// TIA Portal V17 export
// export: Created 2021-12-03T08:13:05.5673976Z, ExportSetting WithDefaults, DisplayName Totally Integrated Automation Portal, DisplayVersion V17, DisplayName TIA Portal Openness, DisplayVersion V17, DisplayName TIA Portal Version Control Interface, DisplayVersion V17, DisplayName STEP 7 Professional, DisplayVersion V17, DisplayName STEP 7 Safety, DisplayVersion V17, DisplayName WinCC Advanced, DisplayVersion V17
FUNCTION "FC_SpdClclt" : Void   // FC503, FBD
VERSION : 0.1
// stored: AutoNumber false, IsIECCheckEnabled false, UDAEnableTagReadback false
   VAR_TEMP
      "Time" : Real;
   END_VAR
   VAR_TEMP   // added for the SCL form of the ladder/FBD networks
      _w1 : Bool;
   END_VAR
BEGIN

REGION Network 1: Условие для запуска
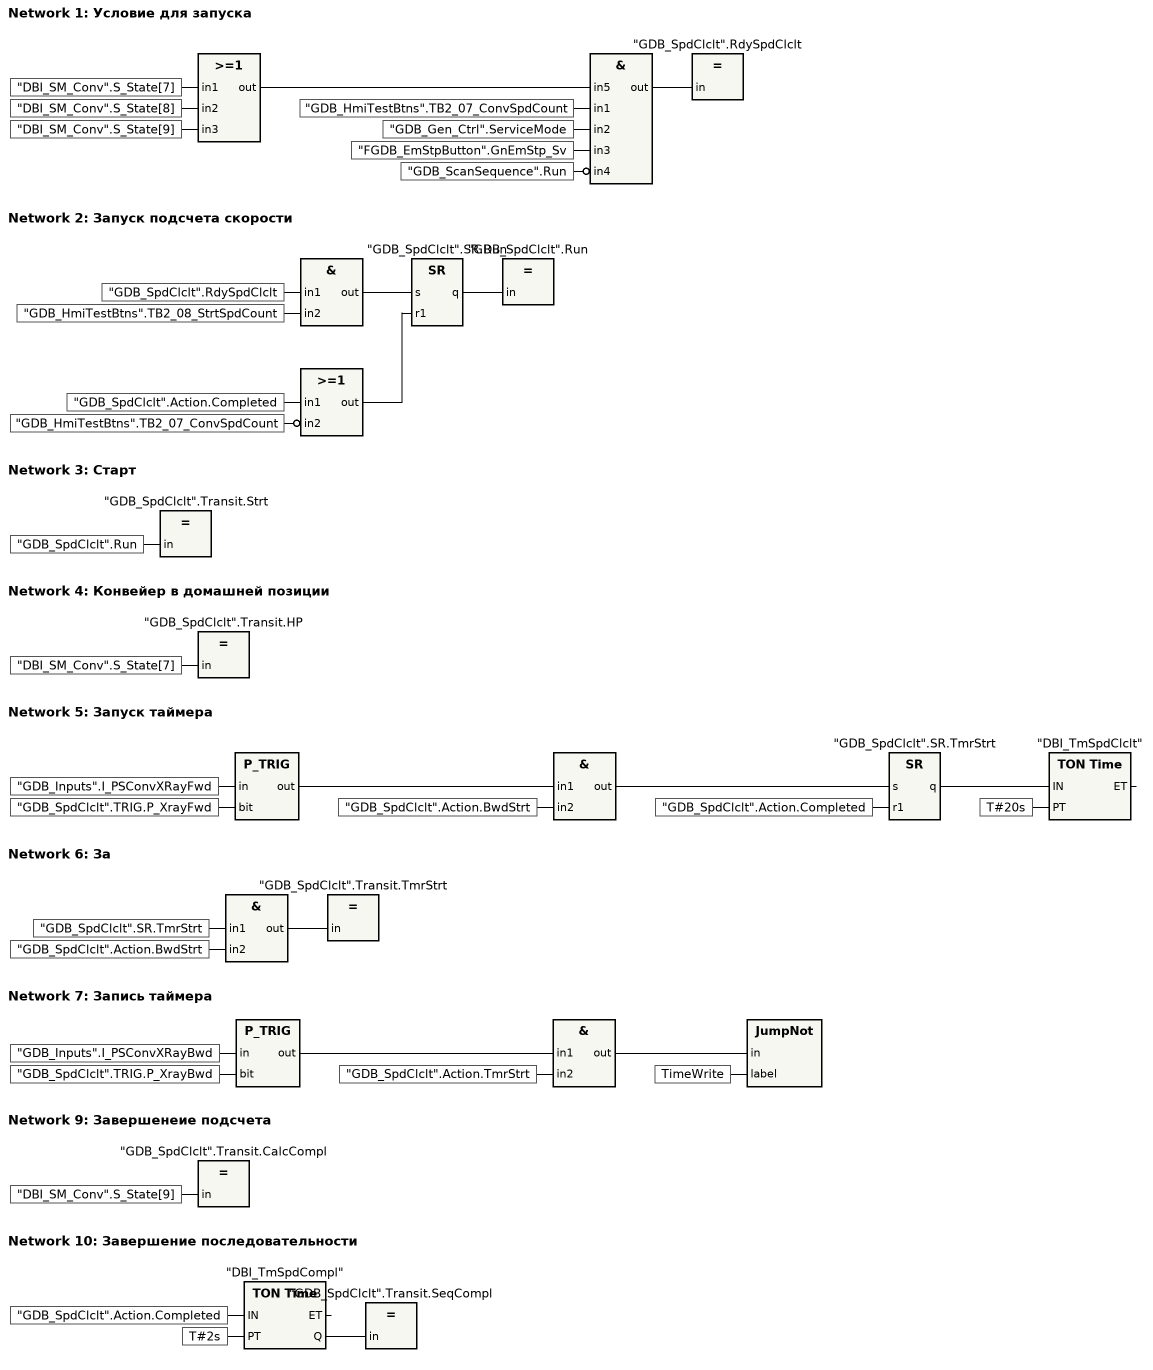
   "GDB_SpdClclt".RdySpdClclt := ("DBI_SM_Conv".S_State[7] OR "DBI_SM_Conv".S_State[8] OR "DBI_SM_Conv".S_State[9]) AND "GDB_HmiTestBtns".TB2_07_ConvSpdCount AND "GDB_Gen_Ctrl".ServiceMode AND "FGDB_EmStpButton".GnEmStp_Sv AND NOT "GDB_ScanSequence".Run;
END_REGION

REGION Network 2: Запуск подсчета скорости
   IF "GDB_SpdClclt".RdySpdClclt AND "GDB_HmiTestBtns".TB2_08_StrtSpdCount THEN
       "GDB_SpdClclt".SR.Run := TRUE;   // SR flip-flop
   END_IF;
   IF "GDB_SpdClclt".Action.Completed OR NOT "GDB_HmiTestBtns".TB2_07_ConvSpdCount THEN
       "GDB_SpdClclt".SR.Run := FALSE;
   END_IF;
   "GDB_SpdClclt".Run := "GDB_SpdClclt".SR.Run;
END_REGION

REGION Network 3: Старт
   "GDB_SpdClclt".Transit.Strt := "GDB_SpdClclt".Run;
END_REGION

REGION Network 4: Конвейер в домашней позиции
   "GDB_SpdClclt".Transit.HP := "DBI_SM_Conv".S_State[7];
END_REGION

REGION Network 5: Запуск таймера
   #_w1 := "GDB_Inputs".I_PSConvXRayFwd AND NOT "GDB_SpdClclt".TRIG.P_XrayFwd;   // rising edge
   "GDB_SpdClclt".TRIG.P_XrayFwd := "GDB_Inputs".I_PSConvXRayFwd;
   IF #_w1 AND "GDB_SpdClclt".Action.BwdStrt THEN
       "GDB_SpdClclt".SR.TmrStrt := TRUE;   // SR flip-flop
   END_IF;
   IF "GDB_SpdClclt".Action.Completed THEN "GDB_SpdClclt".SR.TmrStrt := FALSE; END_IF;
   "DBI_TmSpdClclt".TON(IN := "GDB_SpdClclt".SR.TmrStrt, PT := T#20s);
END_REGION

REGION Network 6: За
   "GDB_SpdClclt".Transit.TmrStrt := "GDB_SpdClclt".SR.TmrStrt AND "GDB_SpdClclt".Action.BwdStrt;
END_REGION

REGION Network 7: Запись таймера
   // no SCL statement known for JumpNot: written as a call
   #_w1 := "GDB_Inputs".I_PSConvXRayBwd AND NOT "GDB_SpdClclt".TRIG.P_XrayBwd;   // rising edge
   "GDB_SpdClclt".TRIG.P_XrayBwd := "GDB_Inputs".I_PSConvXRayBwd;
   JumpNot(in := #_w1 AND "GDB_SpdClclt".Action.TmrStrt, label := TimeWrite);
END_REGION

NETWORK
TITLE = Расчет скорости
      L     "DBI_TmSpdClclt".ET;
      L     1000;
      /R;
      T     #"Time";

      L     "GDB_HMI_IO_Retain".SensDist.DistXRayFwdToXRayBwd;
      L     #"Time";
      /R;
      T     "GDB_SpdClclt".FactSpeed;

      L     "GDB_SpdClclt".FactSpeed;
      T     "GDB_PlcToHmi".Status.FactSpeedCalc;

REGION Network 9: Завершенеие подсчета
   TimeWrite:
   "GDB_SpdClclt".Transit.CalcCompl := "DBI_SM_Conv".S_State[9];
END_REGION

REGION Network 10: Завершение последовательности
   "DBI_TmSpdCompl".TON(IN := "GDB_SpdClclt".Action.Completed, PT := T#2s);
   "GDB_SpdClclt".Transit.SeqCompl := "DBI_TmSpdCompl".Q;
END_REGION

REGION Network 11
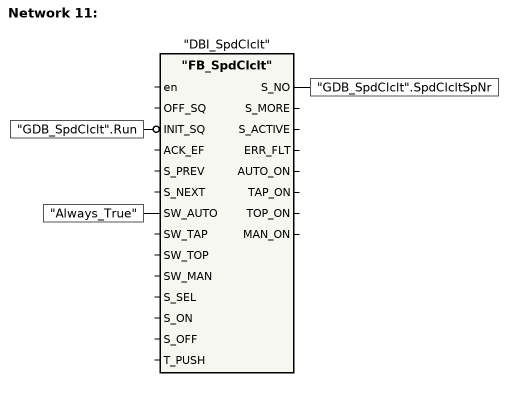
   "DBI_SpdClclt"(INIT_SQ := NOT "GDB_SpdClclt".Run,   // "FB_SpdClclt"
                  SW_AUTO := "Always_True",
                  S_NO => "GDB_SpdClclt".SpdClcltSpNr);
END_REGION
END_FUNCTION
